(* 
:Description:
*)
FUNCTION_BLOCK ABSTRACT FB_UniversalCxUps IMPLEMENTS I_UniversalCxUps
VAR
	bFirstCycle : BOOL := TRUE;
	
	(* Internal parameters *)
	sName 		: STRING;
	sNetID		: STRING;
	iPlcPort 	: UINT;
	tTimeout	: TIME;
	
	(* Internal status *)
	bPowerOk	: BOOL;
END_VAR
(*
Version history:

+-------------+------------+----------------+----------+------------------------------------------+
|Date         | Version    | created under  | Author   | Remark                                   |
+=============+============+================+==========+==========================================+
|2022-01      | 1.0.0.0    | V3.1.4024.22   | ADBO     | Function block created                   |
+-------------+------------+----------------+----------+------------------------------------------+

*)

METHOD MR_FirstCycle : BOOL
VAR_INPUT
	sName 		: STRING;
	sNetID		: STRING;
	iPlcPort 	: UINT;
	tTimeout	: TIME;
END_VAR
THIS^.sName := sName;
THIS^.sNetID := sNetID;
THIS^.iPlcPort := iPlcPort;
THIS^.tTimeout := tTimeout;
END_METHOD

PROPERTY Name : STRING
GET
Name := sName;
END_GET
SET
sName := Name;
END_SET
END_PROPERTY

PROPERTY NetId : STRING
GET
NetId := sNetID;
END_GET
SET
sNetId := NetId;
END_SET
END_PROPERTY

PROPERTY PlcPort : UINT
GET
PlcPort := iPlcPort;
END_GET
SET
iPlcPort := PlcPort;
END_SET
END_PROPERTY

PROPERTY PowerOk : REFERENCE TO BOOL
GET
PowerOk REF= bPowerOk;
END_GET
END_PROPERTY

PROPERTY Timeout : TIME
GET
Timeout := tTimeout;
END_GET
SET
tTimeout := Timeout;
END_SET
END_PROPERTY

END_FUNCTION_BLOCK

(* stored: Version 1.1.0.1, ProductVersion 3.1.4024.9
   POU FB_UniversalCxUps: Id {b494f72d-5973-48b1-87b7-fba9ca370876}, SpecialFunc None
   Folder FirstCycle: Id {ea140722-72f0-433e-82b8-80fa42ec70d2}
   Folder Properties: Id {21af108c-9909-42de-985e-e05dc6fe781a}
   Folder Parameters: Id {7cdc47c0-4de6-4c5f-95bd-1b240c769c9d}
   Folder Status: Id {e3a65237-5693-48aa-b767-a062e86a146a}
   Method MR_FirstCycle: Id {429d4478-8cc1-47b2-bfd1-6fba5029d6c0}
   Property Name: Id {d18b4d08-c699-40d4-98fa-2a5c9546e3a0}
   Get Get: Id {d72c1fdb-89f9-47d9-9adc-b023e71628ee}
   Set Set: Id {ed25cf25-6e9c-4f45-8933-7a27b452cebe}
   Property NetId: Id {cd8e04c2-2b67-4368-ac10-47934fef7e66}
   Get Get: Id {6c394858-0fab-4931-8d9e-2c2013a24b68}
   Set Set: Id {417752e3-ff31-4754-8631-647e7f87f3ac}
   Property PlcPort: Id {029a7380-aabf-47f5-a388-dde141317c89}
   Get Get: Id {f05e89e4-6088-42f9-a2ca-0ca1ed1bc65a}
   Set Set: Id {9a600d95-52b1-4e51-9827-1fcd0b10bcc3}
   Property PowerOk: Id {103db35b-60f7-423c-9a9e-f2692cca72be}
   Get Get: Id {6197fd7d-79e7-41e0-aaa4-2aed5189fd4b}
   Property Timeout: Id {2467ad97-5745-4d0b-b884-61493f209d1b}
   Get Get: Id {b3fe4187-969e-4276-8b8a-4bf4c1937ef8}
   Set Set: Id {0ce70865-9e0c-426c-aa64-2236848c4c67} *)
